// TIA Portal project "MPS 14-01-26" (V18)

(* hardware
DEVICE "S7-1200 station_1"  S7-1200 Station
   slot 0: "Rack_0"  S7-1200 Rack  Rack  V1.0
   slot 1: "MPS"  CPU 1214C DC/DC/DC  6ES7 214-1AG40-0XB0  V4.6
   slot 2: "DI 16x24VDC_1"  6ES7 221-1BH32-0XB0  V2.0
   slot 3: "DQ 16x24VDC_1"  SM 1222 DQ16 x 24VDC  6ES7 222-1BH32-0XB0  V2.0
*)

// ===== PLC "MPS"  CPU 1214C DC/DC/DC =====

VAR_GLOBAL   // PLC tag table "ENTRADAS"
   "S1" AT %I0.0 : Bool;   // BOTAO INICIO
   "B1" AT %I0.1 : Bool;   // sensor peças
END_VAR

FUNCTION "TESTE" : Void   // FC1, LAD
{ S7_Optimized_Access := 'TRUE' }
VERSION : 0.1
BEGIN

REGION Network 1
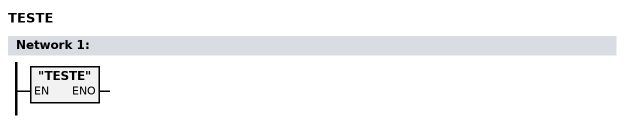
   RUNG wire#powerrail
      "TESTE"()
   END_RUNG
   // the same network as SCL:
   "TESTE"();
END_REGION
END_FUNCTION

FUNCTION "TESTE 2" : Void   // FC2, LAD
{ S7_Optimized_Access := 'TRUE' }
VERSION : 0.1
BEGIN
END_FUNCTION

ORGANIZATION_BLOCK "Main"   // OB1, LAD, ProgramCycle
TITLE = "Main Program Sweep (Cycle)"
{ S7_Optimized_Access := 'TRUE' }
VERSION : 0.1
   VAR_INPUT
      Initial_Call : Bool;   // Initial call of this OB
      Remanence : Bool;   // =True, if remanent data are available
   END_VAR
   VAR_TEMP   // added for the SCL form of the ladder/FBD networks
      _w1 : Bool;
   END_VAR
BEGIN

REGION Network 1
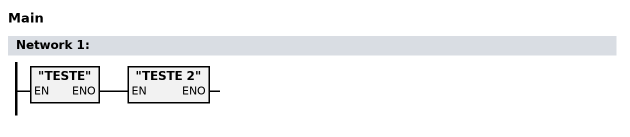
   RUNG wire#powerrail
      "TESTE"()
      "TESTE 2"()
   END_RUNG
   // the same network as SCL:
   "TESTE"(ENO => #_w1);
   IF #_w1 THEN "TESTE 2"(); END_IF;
END_REGION
END_ORGANIZATION_BLOCK